Staubli VAL3: onStart.pgx

public program onStart(string& x_sItem[])
// check and put all the boolean as the status of BIO-MIO-MODBUS-FIELDBUS-ARMIO
  local num i
  local num l_nModbusOut
  local num l_nFieldbusOut
  local bool l_bChange
  local num l_nResult
  local string l_sPath
  local bool l_bCheck
  local string l_sKey
begin
  if x_sItem=="init"
    //
    // DIGITAL INPUT
    //
    // set the default value
    call saveInOut:setInput(0)
//    // BIO
//    call saveInOut:setInput(1)
//    // BIO2 - MIO
//    call saveInOut:setInput(2)
//    // MODBUS
//    call saveInOut:setInput(3)
//    // USER
//    call saveInOut:setInput(4)
//    // REMIO
    //    call saveInOut:setInput(5)
    //.net
    call saveInOut:setInput(6)
    //
    // SAVE
    //
    call save(l_nResult)
    if l_nResult==0
      logMsg("[KERNEL] SUPERVISOR>Input: Save Done")
    else
      logMsg("error "+toString("",l_nResult)+" saving the saveInputInput")
      popUpMsg("error "+toString("",l_nResult)+" saving the saveInputInput")
    endIf
  endIf
  resize(sKey,1,1)
  sKey=""
  if isDefined(saveInOut:dInput["usrIn0"])
    append(sKey)
    sKey[0]="usrIn0"
  endIf
  if isDefined(saveInOut:dInput["usrIn1"])
    append(sKey)
    sKey[1]="usrIn1"
  endIf
  // insert the fIn or usrIn if exist
  if isDefined(saveInOut:dInput["fIn0"])
    sKey[2]="fIn0"
  endIf
  if isDefined(saveInOut:dInput["fIn1"])
    append(sKey)
    sKey[3]="fIn1"
  endIf
  l_sKey=first(saveInOut:dInput)
  i=size(sKey)-1
  //
  // copy all
  //
  while l_sKey!=""
    // use of number
    if find(l_sKey,"fIn")==-1 and find(l_sKey,"usrIn")==-1
      if !(sKey[0]=="" and i==0)
        append(sKey)
        i=i+1
      endIf
      sKey[i]=l_sKey
    endIf
    l_sKey=next(saveInOut:dInput[l_sKey])
  endWhile
end
